Staubli VAL3: TRACK.dtx

public Tracks tTraj{}
  [w]
    frame fFrame = {x=711.850001, y=-407.745087, z=-259.307675, rx=0.000002, ry=0.000003, rz=89.854066, fatherId=world[0]}
    frame fMoving = {x=303.411201, fatherId=tTraj["w"].fFrame[0]}
    num nIndexFrame
    num nIndexTool
    string sID = "w"
    TrajItem tData[3]
      [0]
        num nType
        pointRx pCircle = {fatherId=tTraj["w"].fMoving[0]}
        pointRx pPoint = {fatherId=tTraj["w"].fMoving[0]}
        TrajectoryItem tSuper
          [0]
            string comment = "TRACK ON"
            num distance
            InstrItem iInstr[3]
              [0]
                string sData
                string sType
              [1]
                string sData
                string sType
              [2]
                string sData
                string sType
            num moveType
            num nMoveId
            num nStop
            num nTcpAction
            num nTime
            mdesc nom_speed = {tmax=9999}
            bool toStop
      [1]
        num nType
        pointRx pCircle = {fatherId=tTraj["w"].fMoving[0]}
        pointRx pPoint = {fatherId=tTraj["w"].fMoving[0]}
        TrajectoryItem tSuper
          [0]
            string comment
            num distance
            InstrItem iInstr[3]
              [0]
                string sData
                string sType
              [1]
                string sData
                string sType
              [2]
                string sData
                string sType
            num moveType = 1
            num nMoveId
            num nStop
            num nTcpAction
            num nTime
            mdesc nom_speed = {vel=450, tmax=1000}
            bool toStop
      [2]
        num nType
        pointRx pCircle = {fatherId=tTraj["w"].fMoving[0]}
        pointRx pPoint = {fatherId=tTraj["w"].fMoving[0]}
        TrajectoryItem tSuper
          [0]
            string comment = "TRACK OFF"
            num distance
            InstrItem iInstr[3]
              [0]
                string sData
                string sType
              [1]
                string sData
                string sType
              [2]
                string sData
                string sType
            num moveType
            num nMoveId
            num nStop
            num nTcpAction
            num nTime
            mdesc nom_speed = {tmax=9999}
            bool toStop
